// TIA Portal V20 export
DATA_BLOCK "Instance_FB_IO_Device_Functional_Test_DB"   // DB104
// stored: AutoNumber false, InstanceOfName FB_IO_Device_Functional_Test, InstanceOfType FB
"FB_IO_Device_Functional_Test"
   // VAR_INPUT
   //    Reset_PLC_Functional_Test : Array[0..31] of Bool;
   //    Status : Bool;
   //    Voltage_Read : UInt;
   //    Min_Electrical_Current : UInt;
   //    Max_Electrical_Current : UInt;
   //    Time_End_Electrical_Current_Test : Time;
   //    Time_Start_Visual_Test : Time;
   //    In_Functional_Test_Odd : "IO_Device_Functinal_Test_Odd";
   //    In_Functional_Test_Even : "IO_Device_Functinal_Test_Even";
   // END_VAR
   // VAR_OUTPUT
   //    Out_Test_Parameters_Odd : "IO_Device_Test_Parameters_Odd";
   //    Out_Test_Parameters_Even : "IO_Device_Test_Parameters_Even";
   //    Out_Voltage_Read : UInt;
   //    Comunication_Error_Panel_1 : Bool;
   //    Comunication_Error_Panel_2 : Bool;
   //    Comunication_Error_Panel_3 : Bool;
   //    Comunication_Error_Panel_4 : Bool;
   //    Comunication_Error_Panel_5 : Bool;
   //    Comunication_Error_Panel_6 : Bool;
   //    Comunication_Error_Panel_7 : Bool;
   //    Comunication_Error_Panel_8 : Bool;
   //    Comunication_Error_Panel_9 : Bool;
   //    Comunication_Error_Panel_10 : Bool;
   //    Comunication_Error_Panel_11 : Bool;
   //    Comunication_Error_Panel_12 : Bool;
   //    Comunication_Error_Panel_13 : Bool;
   //    Comunication_Error_Panel_14 : Bool;
   //    Comunication_Error_Panel_15 : Bool;
   //    Comunication_Error_Panel_16 : Bool;
   //    Comunication_Error_Panel_17 : Bool;
   //    Comunication_Error_Panel_18 : Bool;
   //    Comunication_Error_Panel_19 : Bool;
   //    Comunication_Error_Panel_20 : Bool;
   //    Comunication_Error_Panel_21 : Bool;
   //    Comunication_Error_Panel_22 : Bool;
   //    Comunication_Error_Panel_23 : Bool;
   //    Comunication_Error_Panel_24 : Bool;
   //    Comunication_Error_Panel_25 : Bool;
   //    Comunication_Error_Panel_26 : Bool;
   //    Comunication_Error_Panel_27 : Bool;
   //    Comunication_Error_Panel_28 : Bool;
   //    Comunication_Error_Panel_29 : Bool;
   //    Comunication_Error_Panel_30 : Bool;
   // END_VAR
   // VAR
   //    Enable_Comunication_Erro_3 : Bool;
   //    Enable_Comunication_Erro_4 : Bool;
   //    Enable_Comunication_Erro_5 : Bool;
   //    Enable_Comunication_Erro_6 : Bool;
   //    Enable_Comunication_Erro_7 : Bool;
   //    Enable_Comunication_Erro_8 : Bool;
   //    Enable_Comunication_Erro_9 : Bool;
   //    Enable_Comunication_Erro_10 : Bool;
   //    Enable_Comunication_Erro_11 : Bool;
   //    Enable_Comunication_Erro_12 : Bool;
   //    Enable_Comunication_Erro_13 : Bool;
   //    Enable_Comunication_Erro_14 : Bool;
   //    Enable_Comunication_Erro_15 : Bool;
   //    Enable_Comunication_Erro_16 : Bool;
   //    Enable_Comunication_Erro_17 : Bool;
   //    Enable_Comunication_Erro_18 : Bool;
   //    Enable_Comunication_Erro_19 : Bool;
   //    Enable_Comunication_Erro_20 : Bool;
   //    Enable_Comunication_Erro_21 : Bool;
   //    Enable_Comunication_Erro_22 : Bool;
   //    Enable_Comunication_Erro_23 : Bool;
   //    Enable_Comunication_Erro_24 : Bool;
   //    Enable_Comunication_Erro_25 : Bool;
   //    Enable_Comunication_Erro_26 : Bool;
   //    Enable_Comunication_Erro_27 : Bool;
   //    Enable_Comunication_Erro_28 : Bool;
   //    Enable_Comunication_Erro_29 : Bool;
   //    Enable_Comunication_Erro_30 : Bool;
   //    Timer_Alarme_A_1 { S7_SetPoint := 'True'} : TON_TIME;
   //    Timer_Alarme_B_1 { S7_SetPoint := 'True'} : TON_TIME;
   //    Timer_Alarme_A_2 { S7_SetPoint := 'True'} : TON_TIME;
   //    Timer_Alarme_B_2 { S7_SetPoint := 'True'} : TON_TIME;
   //    Timer_Alarme_A_3 { S7_SetPoint := 'True'} : TON_TIME;
   //    Timer_Alarme_B_3 { S7_SetPoint := 'True'} : TON_TIME;
   //    Timer_Alarme_A_4 { S7_SetPoint := 'True'} : TON_TIME;
   //    Timer_Alarme_B_4 { S7_SetPoint := 'True'} : TON_TIME;
   //    Timer_Alarme_A_5 { S7_SetPoint := 'True'} : TON_TIME;
   //    Timer_Alarme_B_5 { S7_SetPoint := 'True'} : TON_TIME;
   //    Timer_Alarme_A_6 { S7_SetPoint := 'True'} : TON_TIME;
   //    Timer_Alarme_B_6 { S7_SetPoint := 'True'} : TON_TIME;
   //    Timer_Alarme_A_7 { S7_SetPoint := 'True'} : TON_TIME;
   //    Timer_Alarme_B_7 { S7_SetPoint := 'True'} : TON_TIME;
   //    Timer_Alarme_A_8 { S7_SetPoint := 'True'} : TON_TIME;
   //    Timer_Alarme_B_8 { S7_SetPoint := 'True'} : TON_TIME;
   //    Timer_Alarme_A_9 { S7_SetPoint := 'True'} : TON_TIME;
   //    Timer_Alarme_B_9 { S7_SetPoint := 'True'} : TON_TIME;
   //    Timer_Alarme_A_10 { S7_SetPoint := 'True'} : TON_TIME;
   //    Timer_Alarme_B_10 { S7_SetPoint := 'True'} : TON_TIME;
   //    Timer_Alarme_A_11 { S7_SetPoint := 'True'} : TON_TIME;
   //    Timer_Alarme_B_11 { S7_SetPoint := 'True'} : TON_TIME;
   //    Timer_Alarme_A_12 { S7_SetPoint := 'True'} : TON_TIME;
   //    Timer_Alarme_B_12 { S7_SetPoint := 'True'} : TON_TIME;
   //    Timer_Alarme_A_13 { S7_SetPoint := 'True'} : TON_TIME;
   //    Timer_Alarme_B_13 { S7_SetPoint := 'True'} : TON_TIME;
   //    Timer_Alarme_A_14 { S7_SetPoint := 'True'} : TON_TIME;
   //    Timer_Alarme_B_14 { S7_SetPoint := 'True'} : TON_TIME;
   //    Timer_Alarme_A_15 { S7_SetPoint := 'True'} : TON_TIME;
   //    Timer_Alarme_B_15 { S7_SetPoint := 'True'} : TON_TIME;
   //    Timer_Alarme_A_16 { S7_SetPoint := 'True'} : TON_TIME;
   //    Timer_Alarme_B_16 { S7_SetPoint := 'True'} : TON_TIME;
   //    Timer_Alarme_A_17 { S7_SetPoint := 'True'} : TON_TIME;
   //    Timer_Alarme_B_17 { S7_SetPoint := 'True'} : TON_TIME;
   //    Timer_Alarme_A_18 { S7_SetPoint := 'True'} : TON_TIME;
   //    Timer_Alarme_B_18 { S7_SetPoint := 'True'} : TON_TIME;
   //    Timer_Alarme_A_19 { S7_SetPoint := 'True'} : TON_TIME;
   //    Timer_Alarme_B_19 { S7_SetPoint := 'True'} : TON_TIME;
   //    Timer_Alarme_A_20 { S7_SetPoint := 'True'} : TON_TIME;
   //    Timer_Alarme_B_20 { S7_SetPoint := 'True'} : TON_TIME;
   //    Timer_Alarme_A_21 { S7_SetPoint := 'True'} : TON_TIME;
   //    Timer_Alarme_B_21 { S7_SetPoint := 'True'} : TON_TIME;
   //    Timer_Alarme_A_22 { S7_SetPoint := 'True'} : TON_TIME;
   //    Timer_Alarme_B_22 { S7_SetPoint := 'True'} : TON_TIME;
   //    Timer_Alarme_A_23 { S7_SetPoint := 'True'} : TON_TIME;
   //    Timer_Alarme_B_23 { S7_SetPoint := 'True'} : TON_TIME;
   //    Timer_Alarme_A_24 { S7_SetPoint := 'True'} : TON_TIME;
   //    Timer_Alarme_B_24 { S7_SetPoint := 'True'} : TON_TIME;
   //    Timer_Alarme_A_25 { S7_SetPoint := 'True'} : TON_TIME;
   //    Timer_Alarme_B_25 { S7_SetPoint := 'True'} : TON_TIME;
   //    Timer_Alarme_A_26 { S7_SetPoint := 'True'} : TON_TIME;
   //    Timer_Alarme_B_26 { S7_SetPoint := 'True'} : TON_TIME;
   //    Timer_Alarme_A_27 { S7_SetPoint := 'True'} : TON_TIME;
   //    Timer_Alarme_B_27 { S7_SetPoint := 'True'} : TON_TIME;
   //    Timer_Alarme_A_28 { S7_SetPoint := 'True'} : TON_TIME;
   //    Timer_Alarme_B_28 { S7_SetPoint := 'True'} : TON_TIME;
   //    Timer_Alarme_A_29 { S7_SetPoint := 'True'} : TON_TIME;
   //    Timer_Alarme_B_29 { S7_SetPoint := 'True'} : TON_TIME;
   //    Timer_Alarme_A_30 { S7_SetPoint := 'True'} : TON_TIME;
   //    Timer_Alarme_B_30 { S7_SetPoint := 'True'} : TON_TIME;
   // END_VAR
BEGIN
END_DATA_BLOCK
